FUNCTION_BLOCK E_CTU
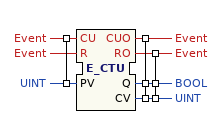
  EVENT_INPUT
    CU WITH PV;
    R;
  END_EVENT
  EVENT_OUTPUT
    CUO WITH Q, CV;
    RO WITH Q, CV;
  END_EVENT
  VAR_INPUT
    PV : UINT;
  END_VAR
  VAR_OUTPUT
    Q : BOOL;
    CV : UINT;
  END_VAR
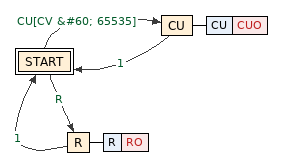
  EC_STATES
    START;
    CU : CU -> CUO;
    R : R -> RO;
  END_STATES
  EC_TRANSITIONS
    START TO CU := CU[CV &#60; 65535];
    CU TO START := 1;
    START TO R := R;
    R TO START := 1;
  END_TRANSITIONS
  ALGORITHM R IN ST:
CV := 0;&#38;#10;Q := FALSE;&#38;#10;
  END_ALGORITHM
  ALGORITHM CU IN ST:
CV := CV + 1;&#38;#10;Q := (CV &#62;= PV);&#38;#10;
  END_ALGORITHM
END_FUNCTION_BLOCK
